(* PLC project Unnamed, Unknown Unnamed 1 *)
(* stored: creationDateTime 2026-06-15T08:02:50, modificationDateTime 2026-06-15T08:02:50 *)

PROGRAM PLC_PRG
  VAR
    blink : BOOL;
    TOF0 : TOF;
    TON0 : TON;
    enable_btn : BOOL;
  END_VAR
  VAR  (* added by the conversion: wires and edge detectors of the diagram *)
    _CURRENT_DT1522858_OUT : ANY;
  END_VAR

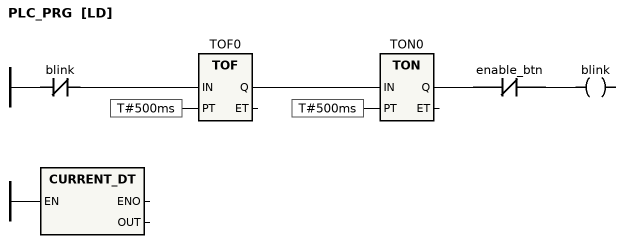
(* LD diagram, written out as Structured Text *)
TOF0(IN := NOT blink, PT := T#500ms);
TON0(IN := TOF0.Q, PT := T#500ms);
blink := TON0.Q AND NOT enable_btn;
_CURRENT_DT1522858_OUT := CURRENT_DT();
END_PROGRAM

CONFIGURATION Config0
  RESOURCE Res0 ON PLC
    TASK task0(INTERVAL := T#20ms, PRIORITY := 1);
    PROGRAM instance0 WITH task0 : PLC_PRG;
  END_RESOURCE
END_CONFIGURATION
